FUNCTION_BLOCK AUDI_TO_AD (* Composite FB for converting AUDI (UDINT) adapter to AD (DWORD) adapter *)
  (* Standard: 61499-2; Description: Copyright (c) 2026 HR Agrartechnik GmbH This program and the accompanying materials are made available under the terms of the Eclipse Public License 2.0 which is available at https://www.eclipse.org/legal/epl-2.0/ SPDX-License-Identifier: EPL-2.0 *)
  (* Version 1.0, 2026-01-17, Franz Höpfinger, HR Agrartechnik GmbH *)
  PACKAGE adapter::conversion::unidirectional;
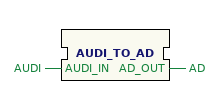
  SOCKETS
    AUDI_IN : adapter::types::unidirectional::AUDI; (* UDINT Adapter Input *)
  END_SOCKETS
  PLUGS
    AD_OUT : adapter::types::unidirectional::AD; (* DWORD Adapter Output *)
  END_PLUGS
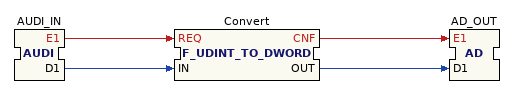
  FBS
    Convert : iec61131::conversion::F_UDINT_TO_DWORD;
  END_FBS
  EVENT_CONNECTIONS
    AUDI_IN.E1 TO Convert.REQ;
    Convert.CNF TO AD_OUT.E1;
  END_CONNECTIONS
  DATA_CONNECTIONS
    AUDI_IN.D1 TO Convert.IN;
    Convert.OUT TO AD_OUT.D1;
  END_CONNECTIONS
END_FUNCTION_BLOCK
